// Mitsubishi GX Works2 project: MPS_0821_실습1   PLC: Q02U

PROGRAM MAIN
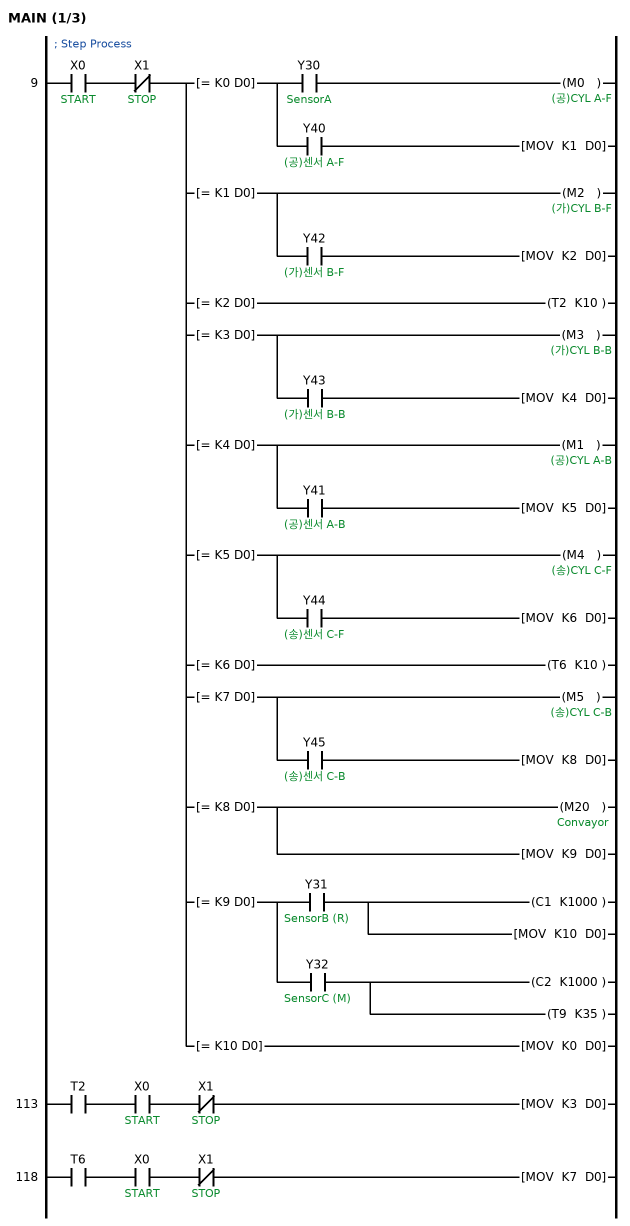
; Step Process
9     LD      X0  ; START
      ANI     X1  ; STOP
      MPS
      AND=    K0 D0
      MPS
      AND     Y30  ; SensorA
      OUT     M0  ; (공)CYL A-F
      MPP
      AND     Y40  ; (공)센서 A-F
      MOV     K1 D0
      MRD
      AND=    K1 D0
      OUT     M2  ; (가)CYL B-F
      AND     Y42  ; (가)센서 B-F
      MOV     K2 D0
      MRD
      AND=    K2 D0
      OUT     T2 K10
      MRD
      AND=    K3 D0
      OUT     M3  ; (가)CYL B-B
      AND     Y43  ; (가)센서 B-B
      MOV     K4 D0
      MRD
      AND=    K4 D0
      OUT     M1  ; (공)CYL A-B
      AND     Y41  ; (공)센서 A-B
      MOV     K5 D0
      MRD
      AND=    K5 D0
      OUT     M4  ; (송)CYL C-F
      AND     Y44  ; (송)센서 C-F
      MOV     K6 D0
      MRD
      AND=    K6 D0
      OUT     T6 K10
      MRD
      AND=    K7 D0
      OUT     M5  ; (송)CYL C-B
      AND     Y45  ; (송)센서 C-B
      MOV     K8 D0
      MRD
      AND=    K8 D0
      OUT     M20  ; Convayor
      MOV     K9 D0
      MRD
      AND=    K9 D0
      MPS
      AND     Y31  ; SensorB (R)
      OUT     C1 K1000
      MOV     K10 D0
      MPP
      AND     Y32  ; SensorC (M)
      OUT     C2 K1000
      OUT     T9 K35
      MPP
      AND=    K10 D0
      MOV     K0 D0
113   LD      T2
      AND     X0  ; START
      ANI     X1  ; STOP
      MOV     K3 D0
118   LD      T6
      AND     X0  ; START
      ANI     X1  ; STOP
      MOV     K7 D0
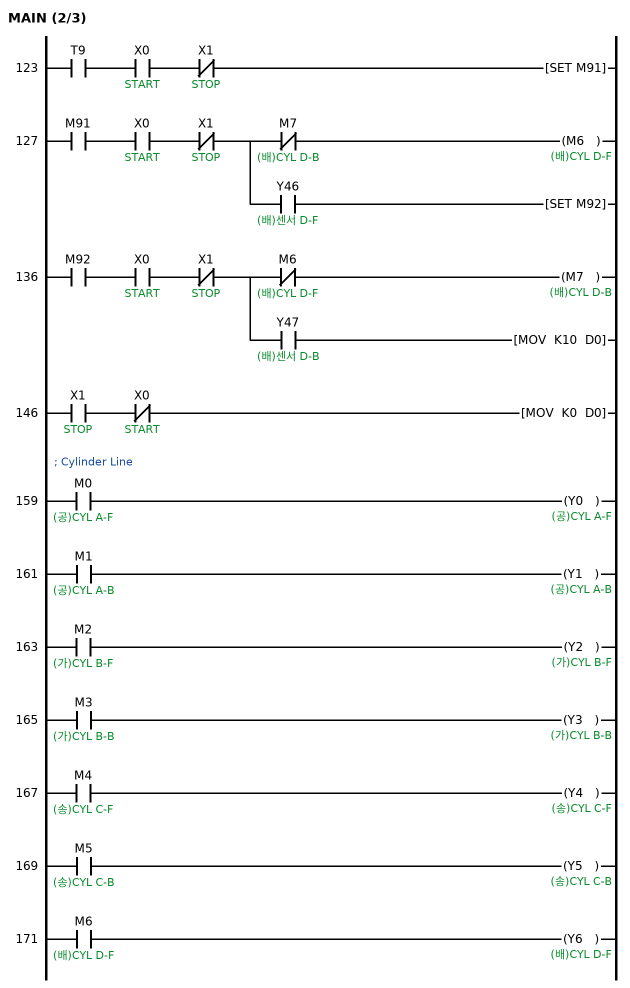
123   LD      T9
      AND     X0  ; START
      ANI     X1  ; STOP
      SET     M91
127   LD      M91
      AND     X0  ; START
      ANI     X1  ; STOP
      MPS
      ANI     M7  ; (배)CYL D-B
      OUT     M6  ; (배)CYL D-F
      MPP
      AND     Y46  ; (배)센서 D-F
      SET     M92
136   LD      M92
      AND     X0  ; START
      ANI     X1  ; STOP
      MPS
      ANI     M6  ; (배)CYL D-F
      OUT     M7  ; (배)CYL D-B
      MPP
      AND     Y47  ; (배)센서 D-B
      MOV     K10 D0
146   LD      X1  ; STOP
      ANI     X0  ; START
      MOV     K0 D0
; Cylinder Line
159   LD      M0  ; (공)CYL A-F
      OUT     Y0  ; (공)CYL A-F
161   LD      M1  ; (공)CYL A-B
      OUT     Y1  ; (공)CYL A-B
163   LD      M2  ; (가)CYL B-F
      OUT     Y2  ; (가)CYL B-F
165   LD      M3  ; (가)CYL B-B
      OUT     Y3  ; (가)CYL B-B
167   LD      M4  ; (송)CYL C-F
      OUT     Y4  ; (송)CYL C-F
169   LD      M5  ; (송)CYL C-B
      OUT     Y5  ; (송)CYL C-B
171   LD      M6  ; (배)CYL D-F
      OUT     Y6  ; (배)CYL D-F
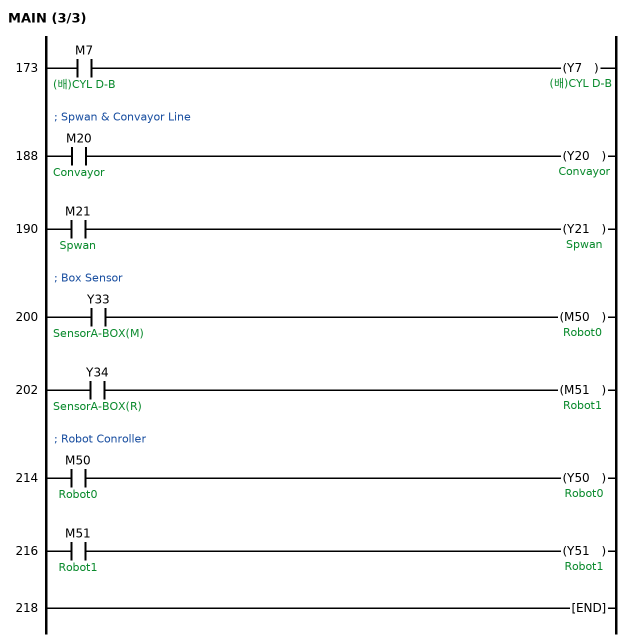
173   LD      M7  ; (배)CYL D-B
      OUT     Y7  ; (배)CYL D-B
; Spwan & Convayor Line
188   LD      M20  ; Convayor
      OUT     Y20  ; Convayor
190   LD      M21  ; Spwan
      OUT     Y21  ; Spwan
; Box Sensor
200   LD      Y33  ; SensorA-BOX(M)
      OUT     M50  ; Robot0
202   LD      Y34  ; SensorA-BOX(R)
      OUT     M51  ; Robot1
; Robot Conroller
214   LD      M50  ; Robot0
      OUT     Y50  ; Robot0
216   LD      M51  ; Robot1
      OUT     Y51  ; Robot1
218   END
END_PROGRAM

// device comments not shown above
X10  ; LAMP(R)
X11  ; LAMP(Y)
X12  ; LAMP(G)
X20  ; Convayor
X21  ; Spwan
Y10  ; RED
Y11  ; YELLOW
Y12  ; GREAN
M10  ; LAMP(R)
M11  ; LAMP(Y)
M12  ; LAMP(G)
M30  ; SensorA
M31  ; SensorB
M32  ; SensorC
M33  ; SensorA-BOX(M)
M34  ; SensorA-BOX(R)
M40  ; (공)센서 A-F
M41  ; (공)센서 A-B
M42  ; (가)센서 B-F
M43  ; (가)센서 B-B
M44  ; (송)센서 C-F
M45  ; (송)센서 C-B
M46  ; (배)센서 D-F
M47  ; (배)센서 D-B
